{attribute 'GeneratedUsingTerminal: EL2502-0010-0020'}
{attribute addProperty BoxType "EL2502-0010-0020"}
{attribute addProperty Id "Activate_permanentBOOL1Activate_DC_start_timeBOOL1DC_ImmediatelyBOOL1ErrAckBOOL1DCSyncOutCh2BOOL1"}
{attribute addProperty CRC "2408987437"}
{attribute addProperty Size "5"}
TYPE Ctrl_8F963B2D :
STRUCT
	{attribute addProperty Name "Activate_permanent"}
	Activate_permanent : BOOL;
	{attribute addProperty Name "Activate_DC_start_time"}
	Activate_DC_start_time : BOOL;
	{attribute addProperty Name "DC_Immediately"}
	DC_Immediately : BOOL;
	{attribute addProperty Name "ErrAck"}
	ErrAck : BOOL;
	{attribute addProperty Name "DCSyncOutCh2"}
	DCSyncOutCh2 : BOOL;
END_STRUCT
END_TYPE

(* stored: Version 1.2.0.0, ProductVersion 3.1.4024.9
   DUT Ctrl_8F963B2D: Id {ffb084fa-ef32-47a3-9f49-f5a59e9968a6} *)
